// Mitsubishi GX Works2 project: Qap-102_E   PLC: Q06H
// MDAS application sample program

PROGRAM Q  // MDAS
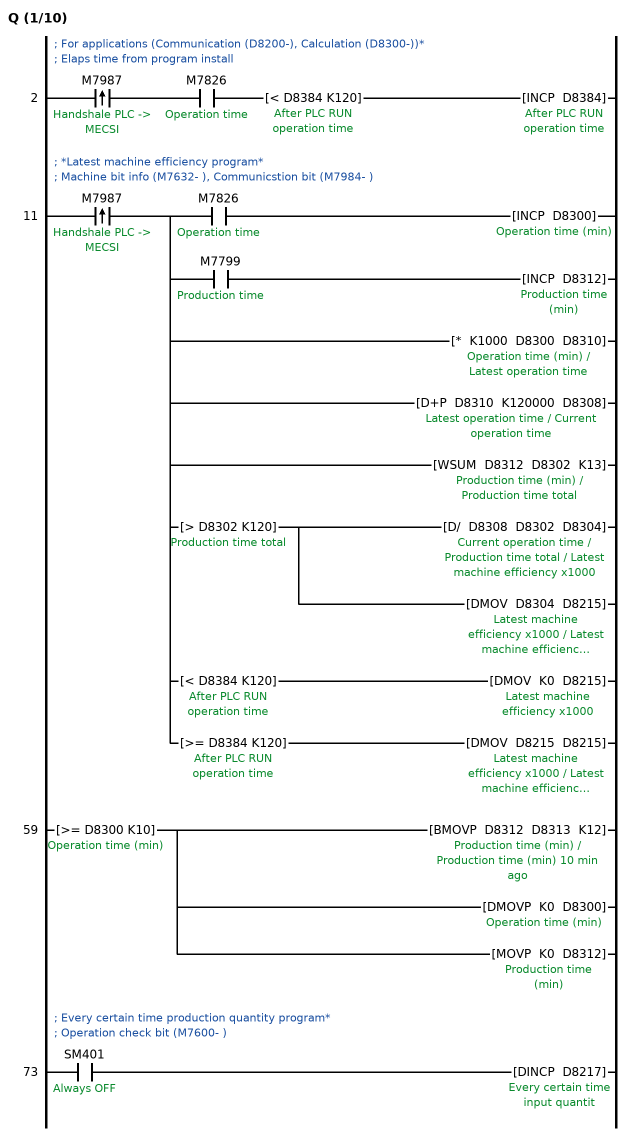
; For applications (Communication (D8200-), Calculation (D8300-))*
; Elaps time from program install
2     LDP     M7987  ; Handshale PLC -> MECSI
      AND     M7826  ; Operation time
      AND<    D8384 K120  ; After PLC RUN operation time
      INCP    D8384
; *Latest machine efficiency program*
; Machine bit info (M7632- ), Communicstion bit (M7984- )
11    LDP     M7987  ; Handshale PLC -> MECSI
      MPS
      AND     M7826  ; Operation time
      INCP    D8300  ; Operation time (min)
      MRD
      AND     M7799  ; Production time
      INCP    D8312  ; Production time (min)
      MPP
      *       K1000 D8300 D8310  ; Latest operation time
      D+P     D8310 K120000 D8308  ; Current operation time
      WSUM    D8312 D8302 K13  ; Production time total
      MPS
      AND>    D8302 K120  ; Production time total
      D/      D8308 D8302 D8304  ; Latest machine efficiency x1000
      DMOV    D8304 D8215  ; Latest machine efficiency x1000
      MRD
      AND<    D8384 K120  ; After PLC RUN operation time
      DMOV    K0 D8215
      MPP
      AND>=   D8384 K120  ; After PLC RUN operation time
      DMOV    D8215 D8215
59    LD>=    D8300 K10  ; Operation time (min)
      BMOVP   D8312 D8313 K12  ; Production time (min) 10 min ago
      DMOVP   K0 D8300
      MOVP    K0 D8312
; Every certain time production quantity program*
; Operation check bit (M7600- )
73    LD      SM401  ; Always OFF
      DINCP   D8217  ; Every certain time input quantit
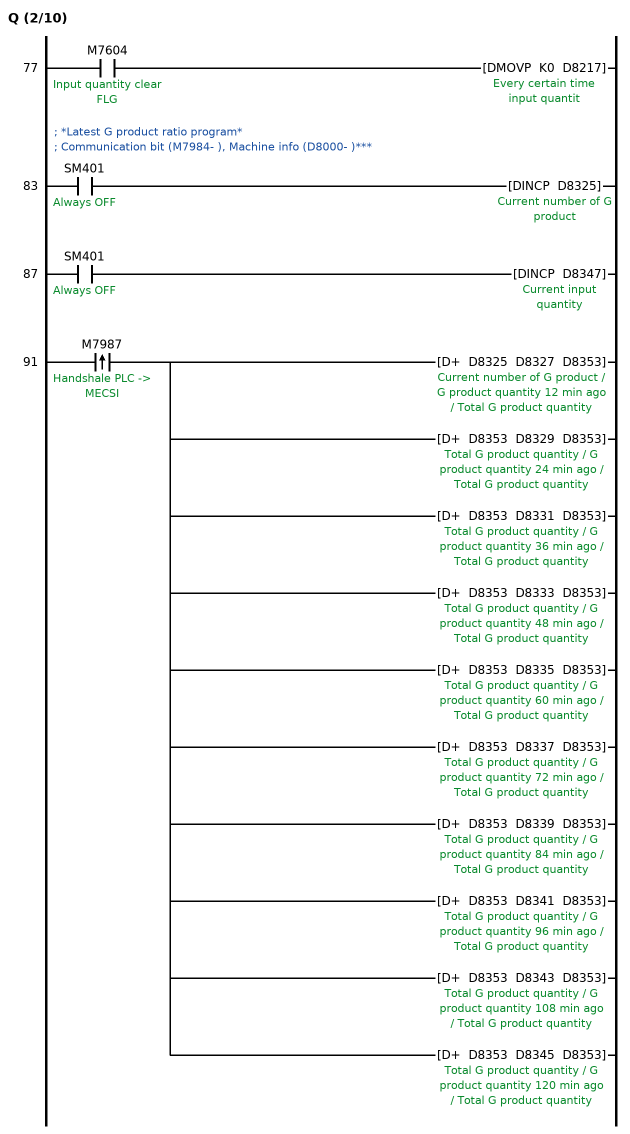
77    LD      M7604  ; Input quantity clear FLG
      DMOVP   K0 D8217
; *Latest G product ratio program*
; Communication bit (M7984- ), Machine info (D8000- )***
83    LD      SM401  ; Always OFF
      DINCP   D8325  ; Current number of G product
87    LD      SM401  ; Always OFF
      DINCP   D8347  ; Current input quantity
91    LDP     M7987  ; Handshale PLC -> MECSI
      D+      D8325 D8327 D8353  ; G product quantity 12 min ago / Total G product quantity
      D+      D8353 D8329 D8353  ; G product quantity 24 min ago
      D+      D8353 D8331 D8353  ; G product quantity 36 min ago
      D+      D8353 D8333 D8353  ; G product quantity 48 min ago
      D+      D8353 D8335 D8353  ; G product quantity 60 min ago
      D+      D8353 D8337 D8353  ; G product quantity 72 min ago
      D+      D8353 D8339 D8353  ; G product quantity 84 min ago
      D+      D8353 D8341 D8353  ; G product quantity 96 min ago
      D+      D8353 D8343 D8353  ; G product quantity 108 min ago
      D+      D8353 D8345 D8353  ; G product quantity 120 min ago
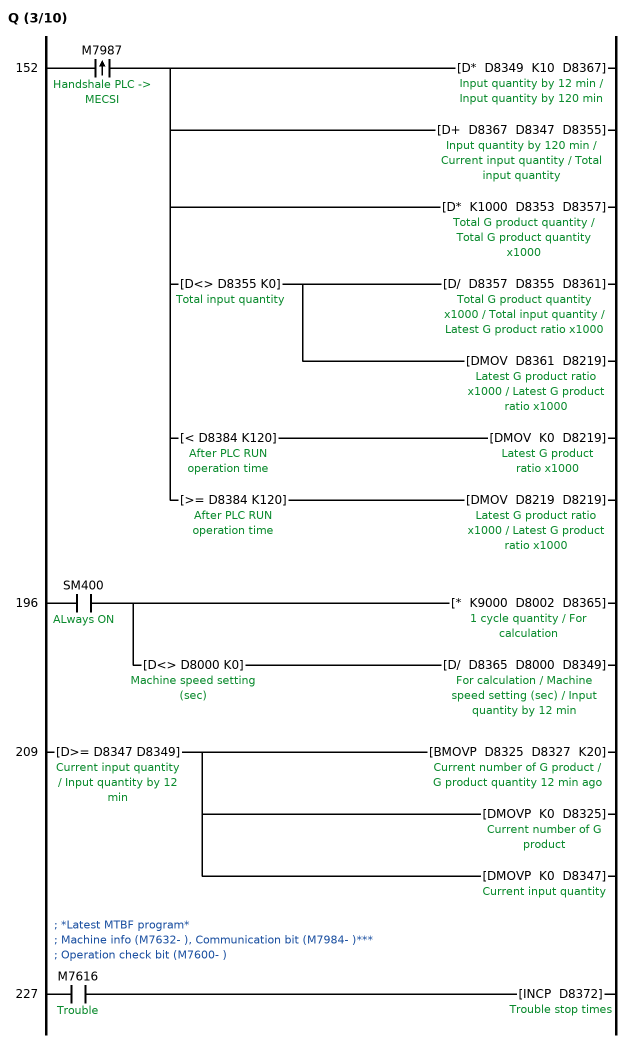
152   LDP     M7987  ; Handshale PLC -> MECSI
      D*      D8349 K10 D8367  ; Input quantity by 12 min / Input quantity by 120 min
      D+      D8367 D8347 D8355  ; Total input quantity
      D*      K1000 D8353 D8357  ; Total G product quantity x1000
      MPS
      ANDD<>  D8355 K0  ; Total input quantity
      D/      D8357 D8355 D8361  ; Latest G product ratio x1000
      DMOV    D8361 D8219  ; Latest G product ratio x1000
      MRD
      AND<    D8384 K120  ; After PLC RUN operation time
      DMOV    K0 D8219
      MPP
      AND>=   D8384 K120  ; After PLC RUN operation time
      DMOV    D8219 D8219
196   LD      SM400  ; ALways ON
      *       K9000 D8002 D8365  ; 1 cycle quantity / For calculation
      ANDD<>  D8000 K0  ; Machine speed setting (sec)
      D/      D8365 D8000 D8349
209   LDD>=   D8347 D8349  ; Current input quantity / Input quantity by 12 min
      BMOVP   D8325 D8327 K20
      DMOVP   K0 D8325
      DMOVP   K0 D8347
; *Latest MTBF program*
; Machine info (M7632- ), Communication bit (M7984- )***
; Operation check bit (M7600- )
227   LD      M7616  ; Trouble
      INCP    D8372  ; Trouble stop times
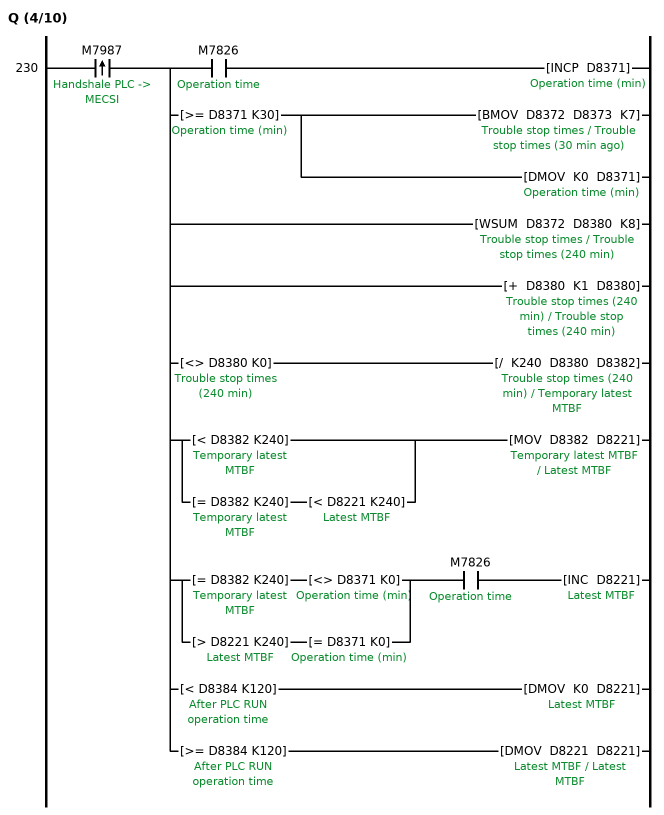
230   LDP     M7987  ; Handshale PLC -> MECSI
      MPS
      AND     M7826  ; Operation time
      INCP    D8371  ; Operation time (min)
      MRD
      AND>=   D8371 K30  ; Operation time (min)
      BMOV    D8372 D8373 K7  ; Trouble stop times (30 min ago)
      DMOV    K0 D8371
      MPP
      WSUM    D8372 D8380 K8  ; Trouble stop times (240 min)
      +       D8380 K1 D8380
      MPS
      AND<>   D8380 K0  ; Trouble stop times (240 min)
      /       K240 D8380 D8382  ; Temporary latest MTBF
      MRD
      LD<     D8382 K240  ; Temporary latest MTBF
      LD=     D8382 K240  ; Temporary latest MTBF
      AND<    D8221 K240  ; Latest MTBF
      ORB
      ANB
      MOV     D8382 D8221
      MRD
      LD=     D8382 K240  ; Temporary latest MTBF
      AND<>   D8371 K0  ; Operation time (min)
      LD>     D8221 K240  ; Latest MTBF
      AND=    D8371 K0  ; Operation time (min)
      ORB
      ANB
      AND     M7826  ; Operation time
      INC     D8221
      MRD
      AND<    D8384 K120  ; After PLC RUN operation time
      DMOV    K0 D8221
      MPP
      AND>=   D8384 K120  ; After PLC RUN operation time
      DMOV    D8221 D8221
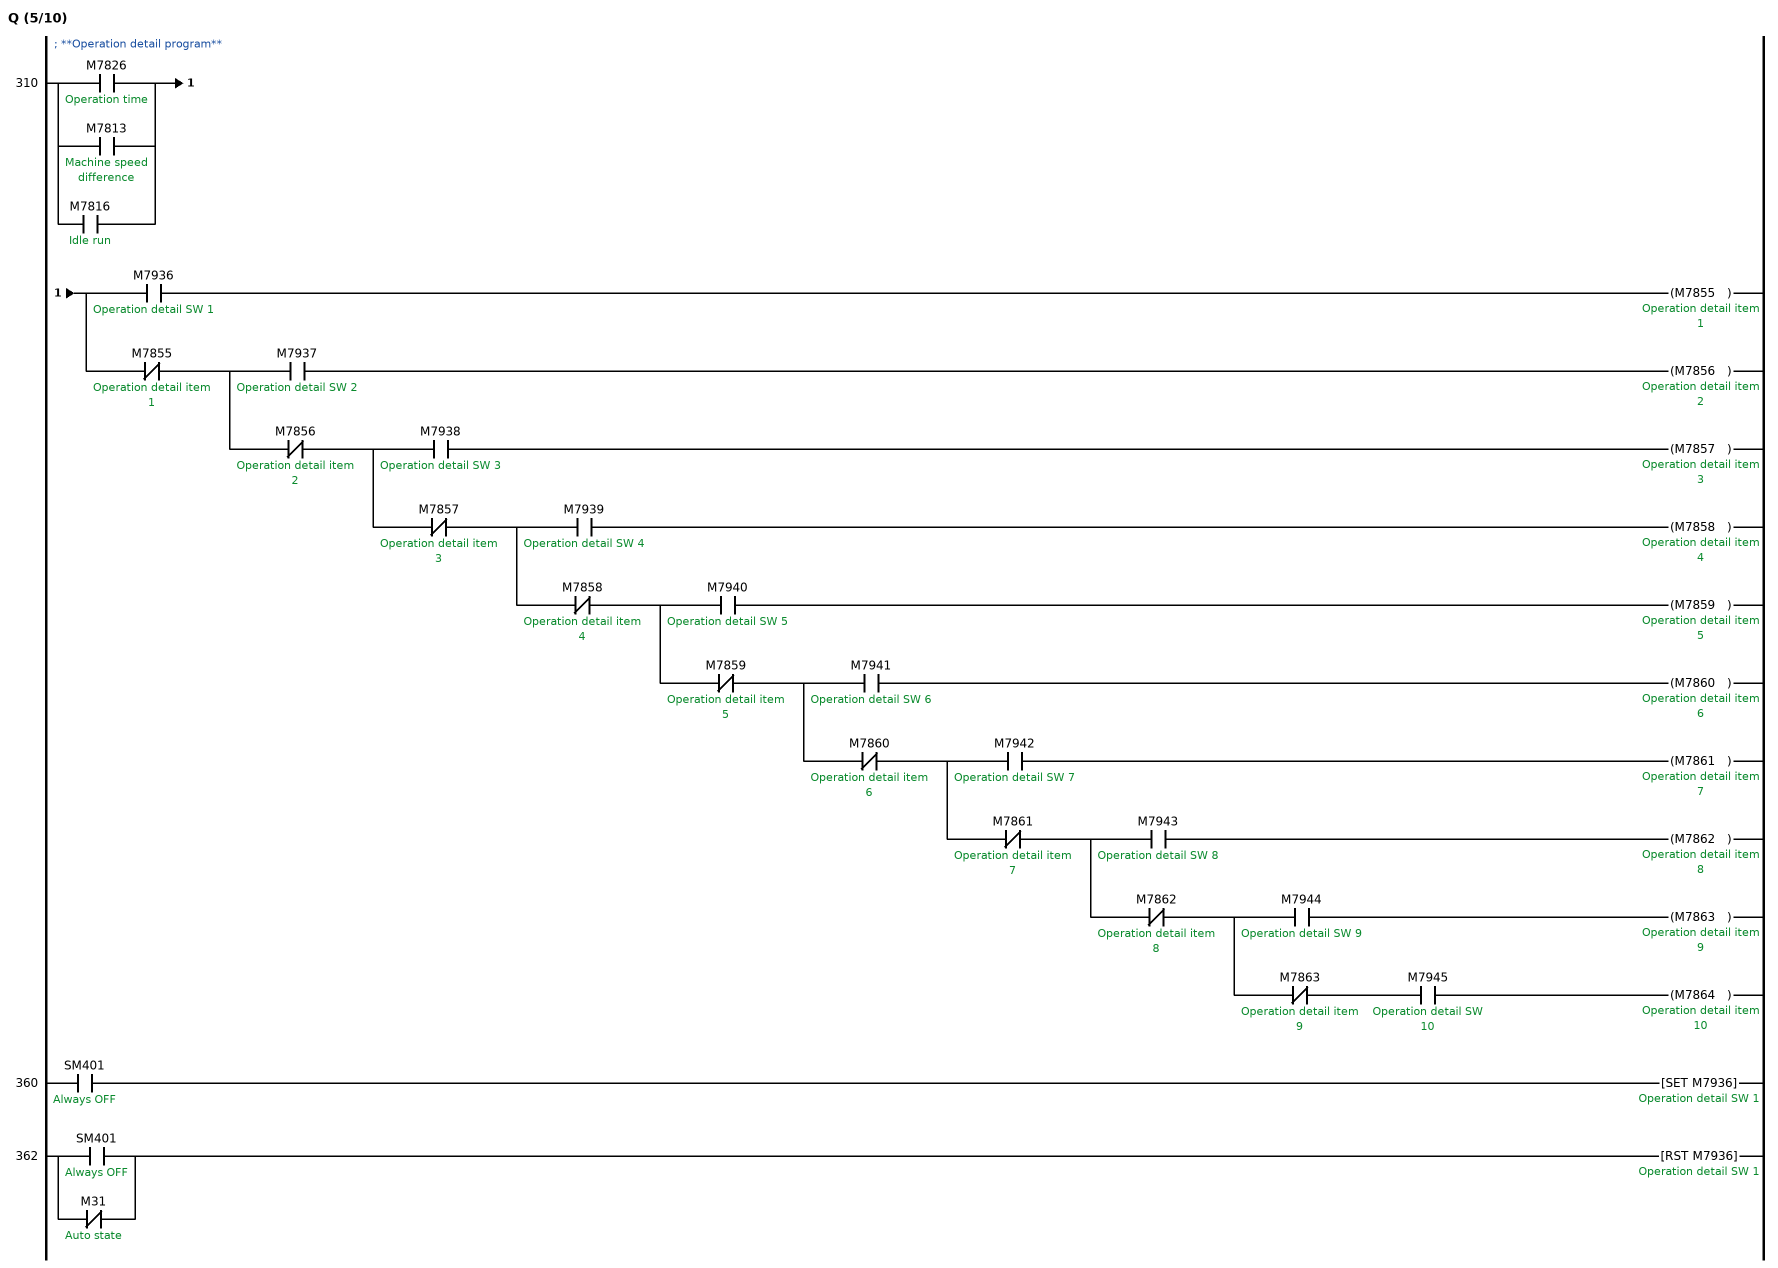
; **Operation detail program**
310   LD      M7826  ; Operation time
      OR      M7813  ; Machine speed difference
      OR      M7816  ; Idle run
      MPS
      AND     M7936  ; Operation detail SW 1
      OUT     M7855  ; Operation detail item 1
      MPP
      ANI     M7855  ; Operation detail item 1
      MPS
      AND     M7937  ; Operation detail SW 2
      OUT     M7856  ; Operation detail item 2
      MPP
      ANI     M7856  ; Operation detail item 2
      MPS
      AND     M7938  ; Operation detail SW 3
      OUT     M7857  ; Operation detail item 3
      MPP
      ANI     M7857  ; Operation detail item 3
      MPS
      AND     M7939  ; Operation detail SW 4
      OUT     M7858  ; Operation detail item 4
      MPP
      ANI     M7858  ; Operation detail item 4
      MPS
      AND     M7940  ; Operation detail SW 5
      OUT     M7859  ; Operation detail item 5
      MPP
      ANI     M7859  ; Operation detail item 5
      MPS
      AND     M7941  ; Operation detail SW 6
      OUT     M7860  ; Operation detail item 6
      MPP
      ANI     M7860  ; Operation detail item 6
      MPS
      AND     M7942  ; Operation detail SW 7
      OUT     M7861  ; Operation detail item 7
      MPP
      ANI     M7861  ; Operation detail item 7
      MPS
      AND     M7943  ; Operation detail SW 8
      OUT     M7862  ; Operation detail item 8
      MPP
      ANI     M7862  ; Operation detail item 8
      MPS
      AND     M7944  ; Operation detail SW 9
      OUT     M7863  ; Operation detail item 9
      MPP
      ANI     M7863  ; Operation detail item 9
      AND     M7945  ; Operation detail SW 10
      OUT     M7864  ; Operation detail item 10
360   LD      SM401  ; Always OFF
      SET     M7936  ; Operation detail SW 1
362   LD      SM401  ; Always OFF
      ORI     M31  ; Auto state
      RST     M7936  ; Operation detail SW 1
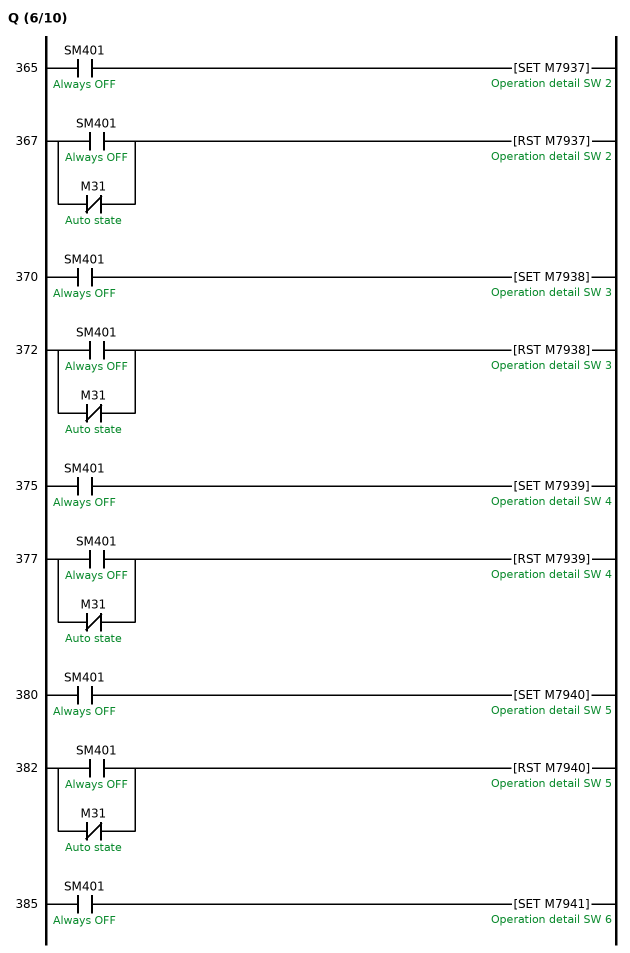
365   LD      SM401  ; Always OFF
      SET     M7937  ; Operation detail SW 2
367   LD      SM401  ; Always OFF
      ORI     M31  ; Auto state
      RST     M7937  ; Operation detail SW 2
370   LD      SM401  ; Always OFF
      SET     M7938  ; Operation detail SW 3
372   LD      SM401  ; Always OFF
      ORI     M31  ; Auto state
      RST     M7938  ; Operation detail SW 3
375   LD      SM401  ; Always OFF
      SET     M7939  ; Operation detail SW 4
377   LD      SM401  ; Always OFF
      ORI     M31  ; Auto state
      RST     M7939  ; Operation detail SW 4
380   LD      SM401  ; Always OFF
      SET     M7940  ; Operation detail SW 5
382   LD      SM401  ; Always OFF
      ORI     M31  ; Auto state
      RST     M7940  ; Operation detail SW 5
385   LD      SM401  ; Always OFF
      SET     M7941  ; Operation detail SW 6
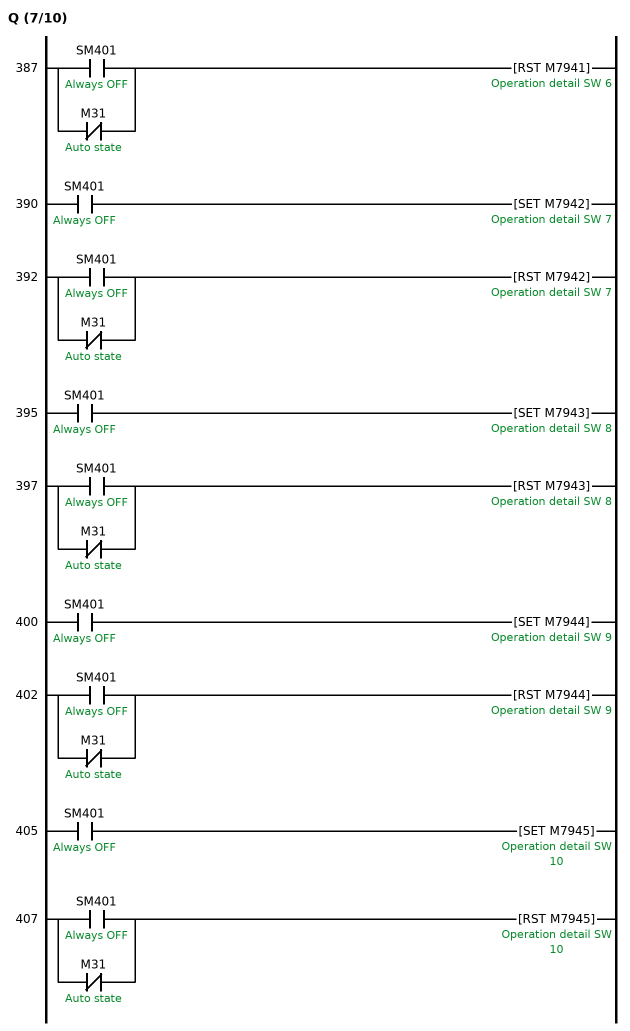
387   LD      SM401  ; Always OFF
      ORI     M31  ; Auto state
      RST     M7941  ; Operation detail SW 6
390   LD      SM401  ; Always OFF
      SET     M7942  ; Operation detail SW 7
392   LD      SM401  ; Always OFF
      ORI     M31  ; Auto state
      RST     M7942  ; Operation detail SW 7
395   LD      SM401  ; Always OFF
      SET     M7943  ; Operation detail SW 8
397   LD      SM401  ; Always OFF
      ORI     M31  ; Auto state
      RST     M7943  ; Operation detail SW 8
400   LD      SM401  ; Always OFF
      SET     M7944  ; Operation detail SW 9
402   LD      SM401  ; Always OFF
      ORI     M31  ; Auto state
      RST     M7944  ; Operation detail SW 9
405   LD      SM401  ; Always OFF
      SET     M7945  ; Operation detail SW 10
407   LD      SM401  ; Always OFF
      ORI     M31  ; Auto state
      RST     M7945  ; Operation detail SW 10
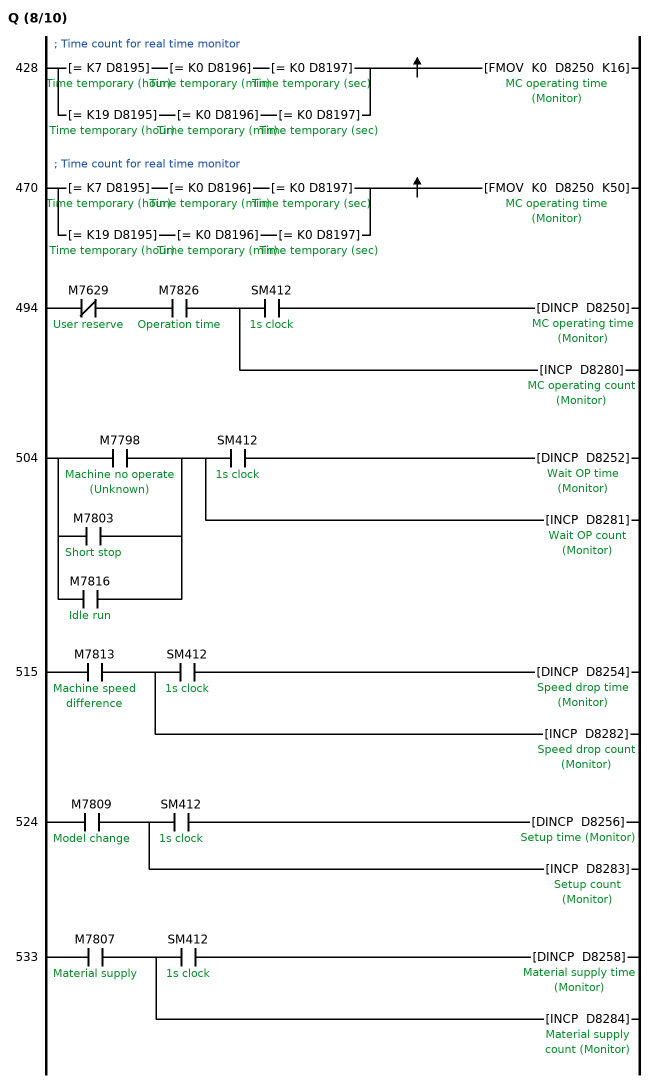
; Time count for real time monitor
428   LD=     K7 D8195  ; Time temporary (hour)
      AND=    K0 D8196  ; Time temporary (min)
      AND=    K0 D8197  ; Time temporary (sec)
      LD=     K19 D8195  ; Time temporary (hour)
      AND=    K0 D8196  ; Time temporary (min)
      AND=    K0 D8197  ; Time temporary (sec)
      ORB
      MEP
      FMOV    K0 D8250 K16  ; MC operating time (Monitor)
; Time count for real time monitor
470   LD=     K7 D8195  ; Time temporary (hour)
      AND=    K0 D8196  ; Time temporary (min)
      AND=    K0 D8197  ; Time temporary (sec)
      LD=     K19 D8195  ; Time temporary (hour)
      AND=    K0 D8196  ; Time temporary (min)
      AND=    K0 D8197  ; Time temporary (sec)
      ORB
      MEP
      FMOV    K0 D8250 K50
494   LDI     M7629  ; User reserve
      AND     M7826  ; Operation time
      MPS
      AND     SM412  ; 1s clock
      DINCP   D8250
      MPP
      INCP    D8280  ; MC operating count (Monitor)
504   LD      M7798  ; Machine no operate (Unknown)
      OR      M7803  ; Short stop
      OR      M7816  ; Idle run
      MPS
      AND     SM412  ; 1s clock
      DINCP   D8252  ; Wait OP time (Monitor)
      MPP
      INCP    D8281  ; Wait OP count (Monitor)
515   LD      M7813  ; Machine speed difference
      MPS
      AND     SM412  ; 1s clock
      DINCP   D8254  ; Speed drop time (Monitor)
      MPP
      INCP    D8282  ; Speed drop count (Monitor)
524   LD      M7809  ; Model change
      MPS
      AND     SM412  ; 1s clock
      DINCP   D8256  ; Setup time (Monitor)
      MPP
      INCP    D8283  ; Setup count (Monitor)
533   LD      M7807  ; Material supply
      MPS
      AND     SM412  ; 1s clock
      DINCP   D8258  ; Material supply time (Monitor)
      MPP
      INCP    D8284  ; Material supply count (Monitor)
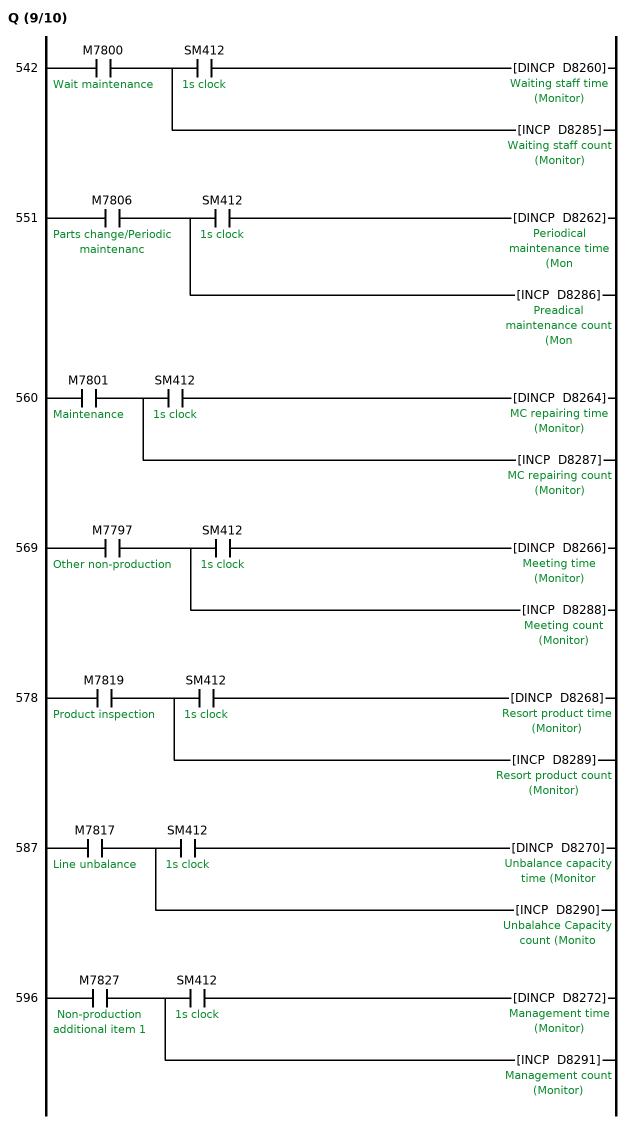
542   LD      M7800  ; Wait maintenance
      MPS
      AND     SM412  ; 1s clock
      DINCP   D8260  ; Waiting staff time (Monitor)
      MPP
      INCP    D8285  ; Waiting staff count (Monitor)
551   LD      M7806  ; Parts change/Periodic maintenanc
      MPS
      AND     SM412  ; 1s clock
      DINCP   D8262  ; Periodical maintenance time (Mon
      MPP
      INCP    D8286  ; Preadical maintenance count (Mon
560   LD      M7801  ; Maintenance
      MPS
      AND     SM412  ; 1s clock
      DINCP   D8264  ; MC repairing time (Monitor)
      MPP
      INCP    D8287  ; MC repairing count (Monitor)
569   LD      M7797  ; Other non-production
      MPS
      AND     SM412  ; 1s clock
      DINCP   D8266  ; Meeting time (Monitor)
      MPP
      INCP    D8288  ; Meeting count (Monitor)
578   LD      M7819  ; Product inspection
      MPS
      AND     SM412  ; 1s clock
      DINCP   D8268  ; Resort product time (Monitor)
      MPP
      INCP    D8289  ; Resort product count (Monitor)
587   LD      M7817  ; Line unbalance
      MPS
      AND     SM412  ; 1s clock
      DINCP   D8270  ; Unbalance capacity time (Monitor
      MPP
      INCP    D8290  ; Unbalahce Capacity count (Monito
596   LD      M7827  ; Non-production additional item 1
      MPS
      AND     SM412  ; 1s clock
      DINCP   D8272  ; Management time (Monitor)
      MPP
      INCP    D8291  ; Management count (Monitor)
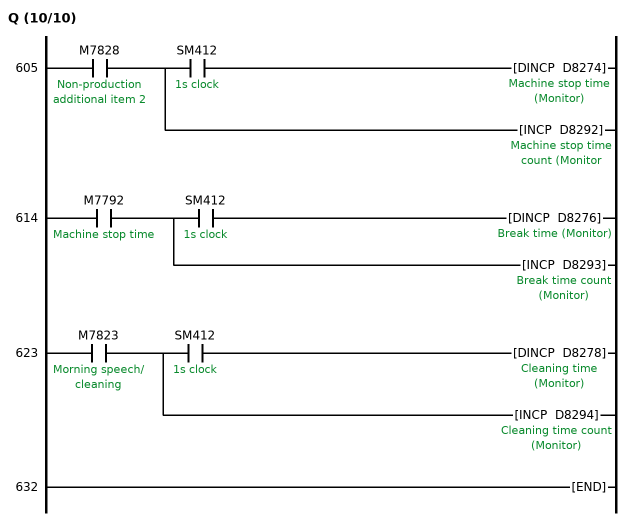
605   LD      M7828  ; Non-production additional item 2
      MPS
      AND     SM412  ; 1s clock
      DINCP   D8274  ; Machine stop time (Monitor)
      MPP
      INCP    D8292  ; Machine stop time count (Monitor
614   LD      M7792  ; Machine stop time
      MPS
      AND     SM412  ; 1s clock
      DINCP   D8276  ; Break time (Monitor)
      MPP
      INCP    D8293  ; Break time count (Monitor)
623   LD      M7823  ; Morning speech/cleaning
      MPS
      AND     SM412  ; 1s clock
      DINCP   D8278  ; Cleaning time (Monitor)
      MPP
      INCP    D8294  ; Cleaning time count (Monitor)
632   END
END_PROGRAM

// device comments not shown above
M7600  ; Operation TRG
M7632  ; Monitor trouble 1
M7984  ; MECSI -> Clear TRG
D8200  ; Lot No.1
